INTERFACE ITcMessage_Ext

METHOD Send : BOOL
VAR_INPUT
	eventType : Tc3_EventLogger.TcEventEntry;
	args : STRING(255);
END_VAR
END_METHOD

END_INTERFACE

(* stored: Version 1.1.0.1, ProductVersion 3.1.4024.11
   Itf ITcMessage_Ext: Id {0257e867-738f-4224-b836-1c0168d03844}
   Method Send: Id {9527ed64-ddfc-4778-91ee-9f9a5b528c9a} *)
